Staubli VAL3: countItem.pjx

--- countItem.pjx ---
Parameters version=s7.2.1 stackSize=5000 millimeterUnit=true
Data file=countItem.dtx

--- countItem.dtx ---
public bool bActive
public string sID
public string sName
public num nCount
public bool bEnable
